TYPE Basic_axis_typ : 	
	STRUCT 
		Input : Basic_Input_typ; (*command structure*)
		Output : Basic_Output_typ; (*parameter structure*)
	END_STRUCT
END_TYPE

(* stored: Version 1.1.0.1, ProductVersion 3.1.4024.3
   DUT Basic_axis_typ: Id {fe209603-205e-0d1c-17d4-f8d0b46b05ba} *)
